// Mitsubishi GX Works2 project: 0624(인터록회로)   PLC: Q02/Q02H

PROGRAM MAIN
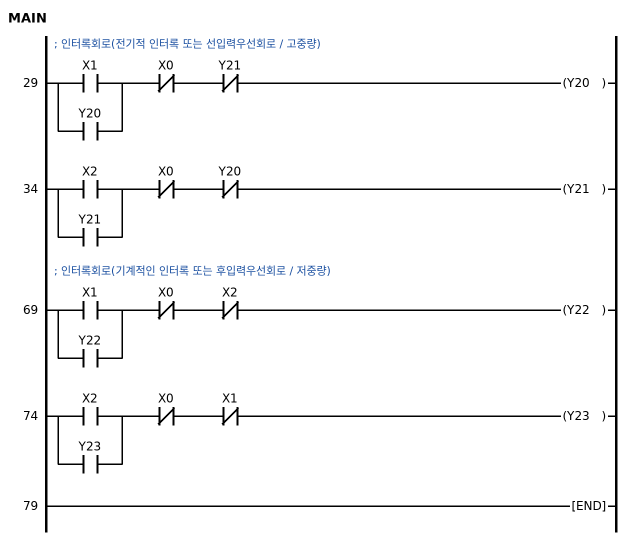
; 인터록회로(전기적 인터록 또는 선입력우선회로 / 고중량)
29    LD      X1
      OR      Y20
      ANI     X0
      ANI     Y21
      OUT     Y20
34    LD      X2
      OR      Y21
      ANI     X0
      ANI     Y20
      OUT     Y21
; 인터록회로(기계적인 인터록 또는 후입력우선회로 / 저중량)
69    LD      X1
      OR      Y22
      ANI     X0
      ANI     X2
      OUT     Y22
74    LD      X2
      OR      Y23
      ANI     X0
      ANI     X1
      OUT     Y23
79    END
END_PROGRAM
